FUNCTION_BLOCK AutomaticCyclicCall EXTENDS Instance IMPLEMENTS I_CyclicInstance
VAR
	membership : AutomaticGlobalInstanceMembership(THIS^);
	_cyclicInstanceCallback : CyclicCallback(0);
END_VAR

PROPERTY PUBLIC CyclicInstanceCallback : I_Callback
GET
CyclicInstanceCallback := _cyclicInstanceCallback;
END_GET
END_PROPERTY

METHOD FB_init : BOOL
VAR_INPUT
	bInitRetains : BOOL; // if TRUE, the retain variables are initialized (warm start / cold start)
	bInCopyCode : BOOL;  // if TRUE, the instance afterwards gets moved into the copy code (online change)
	Target : I_CyclicCalled;
END_VAR
_cyclicInstanceCallback.Target := Target;
END_METHOD

END_FUNCTION_BLOCK

(* stored: Version 1.1.0.1, ProductVersion 3.1.4024.11
   POU AutomaticCyclicCall: Id {a2b7e627-a5fd-402e-9eb5-f07e8064d422}, SpecialFunc None
   Folder Constructor: Id {227b16bd-e892-4d8a-ae22-6c11c5a245f0}
   Property CyclicInstanceCallback: Id {3357174e-c594-4633-a65d-716774e3c184}
   Get Get: Id {2a63e816-aedf-4c00-b118-0232bfc223e2}
   Method FB_init: Id {c65d8418-85fb-461a-ba3b-19538b54bc1a} *)
